FUNCTION RemoveElementFromStringArray : BOOL
VAR_IN_OUT
	arr : ARRAY[*] OF STRING; //must start from 0 index
END_VAR
VAR_INPUT
	target : STRING;
END_VAR
VAR_OUTPUT
	numElements : DINT;
	nextIndex : DINT;
END_VAR
VAR
	i : DINT;
	j : DINT;
END_VAR

FOR i:=LOWER_BOUND(arr, 1) TO UPPER_BOUND(arr, 1) BY 1 DO
	
	IF arr[i] = target THEN
		
		FOR j:=i TO UPPER_BOUND(arr, 1)-1 BY 1 DO
			arr[j] := arr[j+1];
		END_FOR
		
		(*
		MEMMOVE(
			ADR(arr[i]), 
			ADR(arr[ MIN(i+1, UPPER_BOUND(arr, 1)) ]), 
			SIZEOF(STRING) * (UPPER_BOUND(arr, 1) - i) );
		*)
		
		arr[UPPER_BOUND(arr, 1)] := '';
		RemoveElementFromStringArray := TRUE;
		RETURN;

	END_IF
	
END_FOR

END_FUNCTION

(* stored: Version 1.1.0.1, ProductVersion 3.1.4024.11
   POU RemoveElementFromStringArray: Id {5dd27eda-d562-4bc3-bb22-82e5ce25be77}, SpecialFunc None *)
